// TIA Portal V17 export
// export: Created 2025-03-07T09:23:43.6644573Z, ExportSetting WithDefaults, DisplayName Totally Integrated Automation Portal, DisplayVersion V17 Update 8, DisplayName TIA Portal Openness, DisplayVersion V17 Update 8, DisplayName TIA Portal Version Control Interface, DisplayVersion V17, DisplayName SINAMICS Startdrive Advanced, DisplayVersion V17 SP2, DisplayName SINAMICS Startdrive G110M, G120, G120C, G120D, G120P, G115D, DisplayVersion V17 SP2, DisplayName SINAMICS Startdrive G130, G150, S120, S150, SINAMICS MV, S210, DisplayVersion V17 SP2, DisplayName STEP 7 Professional, DisplayVersion V17 Update 8, DisplayName SINUMERIK ONE STEP 7 Toolbox, DisplayVersion V17 Update 12, DisplayName SINUMERIK 840D sl STEP 7 Toolbox, DisplayVersion V17 Update 12, DisplayName STEP 7 Safety, DisplayVersion V17 Update 6, DisplayName WinCC Advanced, DisplayVersion V17 Update 8
FUNCTION "FC2400_GLOBAL_DATA" : Void   // FC2400, LAD
{ S7_Optimized_Access := 'TRUE' }
VERSION : 0.1
// stored: AutoNumber false, IsIECCheckEnabled false, SetENOAutomatically false, UDAEnableTagReadback false
   VAR_TEMP
      RETVAL : Int;
      OPTIONS_ON : Bool;   // OPTIONS ON
      OPTIONS_OFF : Bool;   // OPTIONS OFF
   END_VAR
   VAR_TEMP   // added for the SCL form of the ladder/FBD networks
      _w1 : Bool;
   END_VAR
BEGIN

REGION Network 1: OPTIONS OFF
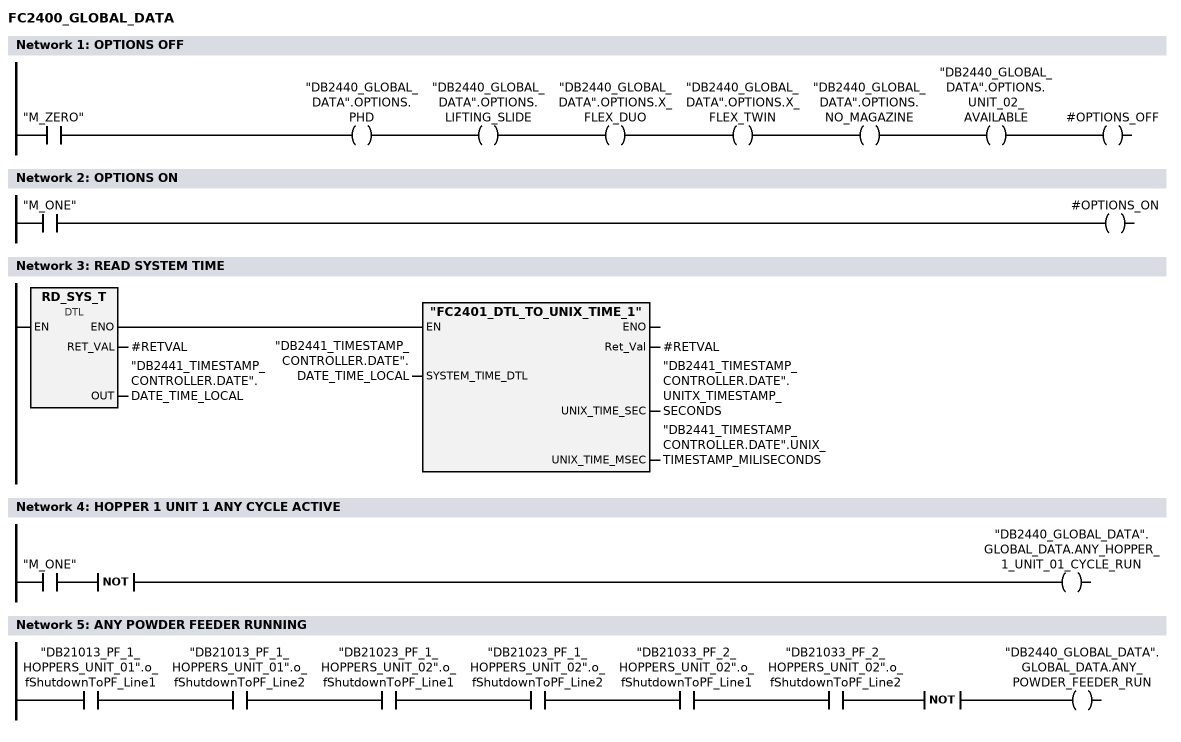
   RUNG wire#powerrail
      Contact( "M_ZERO" )
      Coil( "DB2440_GLOBAL_DATA".OPTIONS.PHD )
      Coil( "DB2440_GLOBAL_DATA".OPTIONS.LIFTING_SLIDE )
      Coil( "DB2440_GLOBAL_DATA".OPTIONS.X_FLEX_DUO )
      Coil( "DB2440_GLOBAL_DATA".OPTIONS.X_FLEX_TWIN )
      Coil( "DB2440_GLOBAL_DATA".OPTIONS.NO_MAGAZINE )
      Coil( "DB2440_GLOBAL_DATA".OPTIONS.UNIT_02_AVAILABLE )
      Coil( #OPTIONS_OFF )
   END_RUNG
   // the same network as SCL:
   "DB2440_GLOBAL_DATA".OPTIONS.PHD := "M_ZERO";
   "DB2440_GLOBAL_DATA".OPTIONS.LIFTING_SLIDE := "M_ZERO";
   "DB2440_GLOBAL_DATA".OPTIONS.X_FLEX_DUO := "M_ZERO";
   "DB2440_GLOBAL_DATA".OPTIONS.X_FLEX_TWIN := "M_ZERO";
   "DB2440_GLOBAL_DATA".OPTIONS.NO_MAGAZINE := "M_ZERO";
   "DB2440_GLOBAL_DATA".OPTIONS.UNIT_02_AVAILABLE := "M_ZERO";
   #OPTIONS_OFF := "M_ZERO";
END_REGION

REGION Network 2: OPTIONS ON
   RUNG wire#powerrail
      Contact( "M_ONE" )
      Coil( #OPTIONS_ON )
   END_RUNG
   // the same network as SCL:
   #OPTIONS_ON := "M_ONE";
END_REGION

REGION Network 3: READ SYSTEM TIME
   RUNG wire#powerrail
      { S7_Templates := "date_type := DTL" } RD_SYS_T(RET_VAL => #RETVAL, OUT => "DB2441_TIMESTAMP_CONTROLLER.DATE".DATE_TIME_LOCAL)
      "FC2401_DTL_TO_UNIX_TIME_1"(SYSTEM_TIME_DTL := "DB2441_TIMESTAMP_CONTROLLER.DATE".DATE_TIME_LOCAL, Ret_Val => #RETVAL, UNIX_TIME_SEC => "DB2441_TIMESTAMP_CONTROLLER.DATE".UNITX_TIMESTAMP_SECONDS, UNIX_TIME_MSEC => "DB2441_TIMESTAMP_CONTROLLER.DATE".UNIX_TIMESTAMP_MILISECONDS)
   END_RUNG
   // the same network as SCL:
   #RETVAL := RD_SYS_T(OUT => "DB2441_TIMESTAMP_CONTROLLER.DATE".DATE_TIME_LOCAL, ENO => #_w1);
   IF #_w1 THEN
       #RETVAL := "FC2401_DTL_TO_UNIX_TIME_1"(SYSTEM_TIME_DTL := "DB2441_TIMESTAMP_CONTROLLER.DATE".DATE_TIME_LOCAL,
                               UNIX_TIME_SEC => "DB2441_TIMESTAMP_CONTROLLER.DATE".UNITX_TIMESTAMP_SECONDS,
                               UNIX_TIME_MSEC => "DB2441_TIMESTAMP_CONTROLLER.DATE".UNIX_TIMESTAMP_MILISECONDS);
   END_IF;
END_REGION

REGION Network 4: HOPPER 1 UNIT 1 ANY CYCLE ACTIVE
   RUNG wire#powerrail
      Contact( "M_ONE" )
      Not()
      Coil( "DB2440_GLOBAL_DATA".GLOBAL_DATA.ANY_HOPPER_1_UNIT_01_CYCLE_RUN )
   END_RUNG
   // the same network as SCL:
   "DB2440_GLOBAL_DATA".GLOBAL_DATA.ANY_HOPPER_1_UNIT_01_CYCLE_RUN := NOT "M_ONE";
END_REGION

REGION Network 5: ANY POWDER FEEDER RUNNING
   RUNG wire#powerrail
      Contact( "DB21013_PF_1_HOPPERS_UNIT_01".o_fShutdownToPF_Line1 )
      Contact( "DB21013_PF_1_HOPPERS_UNIT_01".o_fShutdownToPF_Line2 )
      Contact( "DB21023_PF_1_HOPPERS_UNIT_02".o_fShutdownToPF_Line1 )
      Contact( "DB21023_PF_1_HOPPERS_UNIT_02".o_fShutdownToPF_Line2 )
      Contact( "DB21033_PF_2_HOPPERS_UNIT_02".o_fShutdownToPF_Line1 )
      Contact( "DB21033_PF_2_HOPPERS_UNIT_02".o_fShutdownToPF_Line2 )
      Not()
      Coil( "DB2440_GLOBAL_DATA".GLOBAL_DATA.ANY_POWDER_FEEDER_RUN )
   END_RUNG
   // the same network as SCL:
   "DB2440_GLOBAL_DATA".GLOBAL_DATA.ANY_POWDER_FEEDER_RUN := NOT ("DB21013_PF_1_HOPPERS_UNIT_01".o_fShutdownToPF_Line1 AND "DB21013_PF_1_HOPPERS_UNIT_01".o_fShutdownToPF_Line2 AND "DB21023_PF_1_HOPPERS_UNIT_02".o_fShutdownToPF_Line1 AND "DB21023_PF_1_HOPPERS_UNIT_02".o_fShutdownToPF_Line2 AND "DB21033_PF_2_HOPPERS_UNIT_02".o_fShutdownToPF_Line1 AND "DB21033_PF_2_HOPPERS_UNIT_02".o_fShutdownToPF_Line2);
END_REGION
END_FUNCTION
